FUNCTION_BLOCK FbSimMotorGear (* Виртуальный МЭО для отладки шагового регулятора. *)
  (* Standard: 61499-1; Description: Виртуальный МЭО для отладки шагового регулятора. Simple FB with one algorithm *)
  (* Version 0.2, 2026-03-20, VA, LIB_PLC *)
  (* Documentation:
  // Виртуальный МЭО для отладки шагового регулятора. //           DbSimMotorGear //    +--------------------------+ //    |      FbSimMotorGear      | // ->-|CmdOpen           Position|->- // ->-|CmdClose        SensorOpen|- //   -|TimeOpen       SensorClose|- //   -|TimeClose                 | //   -|Ts                        | //   -|Reset                     | //    +--------------------------+
  *)
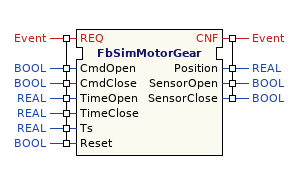
  EVENT_INPUT
    REQ WITH CmdOpen, CmdClose, TimeOpen, TimeClose, Ts, Reset; (* Normal Execution Request *)
  END_EVENT
  EVENT_OUTPUT
    CNF WITH Position, SensorOpen, SensorClose; (* Execution Confirmation *)
  END_EVENT
  VAR_INPUT
    CmdOpen : BOOL := FALSE;
    CmdClose : BOOL := FALSE;
    TimeOpen : REAL := 60.0;
    TimeClose : REAL := 50.0;
    Ts : REAL := 0.1;
    Reset : BOOL := FALSE;
  END_VAR
  VAR_OUTPUT
    Position : REAL := 0.0;
    SensorOpen : BOOL := FALSE;
    SensorClose : BOOL := FALSE;
  END_VAR
  VAR
    SpeedPos : REAL := 0.0; (* Скорость открытия. *)
    SpeedNeg : REAL := 0.0; (* Скорость закрытия. *)
  END_VAR
  EC_STATES
    REQ : REQ -> CNF;
  END_STATES
  ALGORITHM REQ IN ST:
IF(Reset) THEN
	Position := 0.0;
END_IF;

SpeedPos := 100.0 / TimeOpen; // [%/s]
SpeedNeg := 100.0 / TimeClose; // [%/s]

IF(CmdOpen) THEN
	Position := Position + SpeedPos * Ts; // [%]
END_IF;

IF(CmdClose) THEN
	Position := Position - SpeedNeg * Ts; // [%]
END_IF;

IF(Position >= 100.0) THEN
	Position := 100.0;
	SensorOpen := TRUE;
ELSE
	SensorOpen := FALSE;
END_IF;

IF(Position <= 0.0) THEN
	Position := 0.0;
	SensorClose := TRUE;
ELSE
	SensorClose := FALSE;
END_IF;

// @COPYLEFT ALL WRONGS RESERVED :)
// Author: VA
// Contacts: DIY.PLC.314@gmail.com
// Date start LIB_PLC: 2014
// License: GNU GPL-2.0-or-later
// https://www.gnu.org/licenses/old-licenses/gpl-2.0.html
// https://www.youtube.com/watch?v=n1F_MfLRlX0
// https://www.youtube.com/@DIY_PLC
// https://github.com/DIYPLC/LIB_PLC
// https://oshwlab.com/diy.plc.314/PLC_HW1_SW1
// https://3dtoday.ru/3d-models/mechanical-parts/body/korpus-na-din-reiku
// https://t.me/DIY_PLC
  END_ALGORITHM
END_FUNCTION_BLOCK
